// TIA Portal V21 export
TYPE "lubricationSystemStopCtx"
   STRUCT
      "step" : USInt;
      stepTime : LTime;
      alm : "lubricationSystemAlm";
      almDWord { S7_SetPoint := 'True'} : DWord;
   END_STRUCT;
END_TYPE
